// TIA Portal V20 export
FUNCTION "DemoIdentRf" : Void   // FC39, LAD
TITLE = Demo: Ident
AUTHOR : SICAR
FAMILY : Demo
VERSION : 1.0
// Demo for usage of ident moduls
// stored: IsIECCheckEnabled true, SetENOAutomatically true
   // Ret_Val : Ret_Val
BEGIN

REGION Network 1: ChangeLog
   // Change log table:
   // Version | Date | Expert in charge | Changes applied
   // -------|---------|-------------|--------------------------------------------
   // 05.00.00 | 01.09.2023 | SICAR | First released version
END_REGION

REGION Network 2: Define reading informations
   // Write the String "Siemens" in the writting structur of the FB
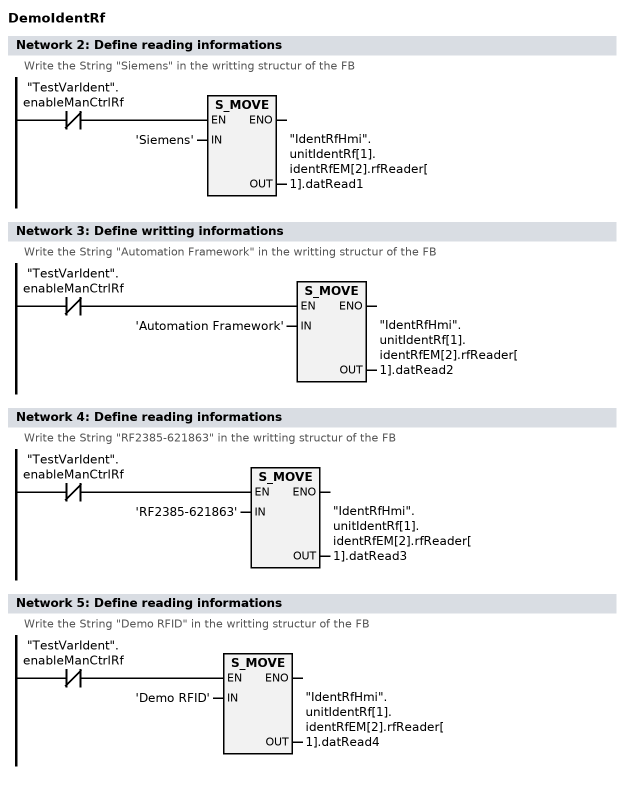
   RUNG wire#powerrail
      I_Contact( "TestVarIdent".enableManCtrlRf )
      S_Move(in := 'Siemens', out => "IdentRfHmi".unitIdentRf[1].identRfEM[2].rfReader[1].datRead1)
   END_RUNG
   // the same network as SCL:
   IF NOT "TestVarIdent".enableManCtrlRf THEN
       "IdentRfHmi".unitIdentRf[1].identRfEM[2].rfReader[1].datRead1 := 'Siemens';
   END_IF;
END_REGION

REGION Network 3: Define writting informations
   // Write the String "Automation Framework" in the writting structur of the FB
   RUNG wire#powerrail
      I_Contact( "TestVarIdent".enableManCtrlRf )
      S_Move(in := 'Automation Framework', out => "IdentRfHmi".unitIdentRf[1].identRfEM[2].rfReader[1].datRead2)
   END_RUNG
   // the same network as SCL:
   IF NOT "TestVarIdent".enableManCtrlRf THEN
       "IdentRfHmi".unitIdentRf[1].identRfEM[2].rfReader[1].datRead2 := 'Automation Framework';
   END_IF;
END_REGION

REGION Network 4: Define reading informations
   // Write the String "RF2385-621863" in the writting structur of the FB
   RUNG wire#powerrail
      I_Contact( "TestVarIdent".enableManCtrlRf )
      S_Move(in := 'RF2385-621863', out => "IdentRfHmi".unitIdentRf[1].identRfEM[2].rfReader[1].datRead3)
   END_RUNG
   // the same network as SCL:
   IF NOT "TestVarIdent".enableManCtrlRf THEN
       "IdentRfHmi".unitIdentRf[1].identRfEM[2].rfReader[1].datRead3 := 'RF2385-621863';
   END_IF;
END_REGION

REGION Network 5: Define reading informations
   // Write the String "Demo RFID" in the writting structur of the FB
   RUNG wire#powerrail
      I_Contact( "TestVarIdent".enableManCtrlRf )
      S_Move(in := 'Demo RFID', out => "IdentRfHmi".unitIdentRf[1].identRfEM[2].rfReader[1].datRead4)
   END_RUNG
   // the same network as SCL:
   IF NOT "TestVarIdent".enableManCtrlRf THEN
       "IdentRfHmi".unitIdentRf[1].identRfEM[2].rfReader[1].datRead4 := 'Demo RFID';
   END_IF;
END_REGION
END_FUNCTION
